TYPE ST_OpModes :
STRUCT
	Standby: BOOL;
	Auto: BOOL;
	Manual: BOOL;
	MDI: BOOL;
	///Reference		: BOOL;  TC3HR
	Homing: BOOL;
END_STRUCT
END_TYPE

(* stored: Version 1.1.0.1, ProductVersion 3.1.0.12
   DUT ST_OpModes: Id {ce08ea52-1088-4cb3-81a1-8f95ccb3ece5} *)
